   PRODUCT_TYPE[1].Motion.Ring_Turntable_Axis_2.Position[8].Pos := 318501;
   PRODUCT_TYPE[1].Motion.Ring_Turntable_Axis_2.Position[8].Vel := 10000;
   PRODUCT_TYPE[2].Motion.Ring_Turntable_Axis_2.Position[8].Pos := 318501;
   PRODUCT_TYPE[2].Motion.Ring_Turntable_Axis_2.Position[8].Vel := 10000;
   PRODUCT_TYPE[3].Motion.Ring_Turntable_Axis_2.Position[8].Pos := 318501;
   PRODUCT_TYPE[3].Motion.Ring_Turntable_Axis_2.Position[8].Vel := 10000;
   PRODUCT_TYPE[4].Motion.Ring_Turntable_Axis_2.Position[8].Pos := 318501;
   PRODUCT_TYPE[4].Motion.Ring_Turntable_Axis_2.Position[8].Vel := 10000;
   PRODUCT_TYPE[5].Motion.Ring_Turntable_Axis_2.Position[8].Pos := 318501;
   PRODUCT_TYPE[5].Motion.Ring_Turntable_Axis_2.Position[8].Vel := 10000;
   PRODUCT_TYPE[6].Motion.Ring_Turntable_Axis_2.Position[8].Pos := 318501;
   PRODUCT_TYPE[6].Motion.Ring_Turntable_Axis_2.Position[8].Vel := 10000;
   PRODUCT_TYPE[7].Motion.Ring_Turntable_Axis_2.Position[8].Pos := 318501;
   PRODUCT_TYPE[7].Motion.Ring_Turntable_Axis_2.Position[8].Vel := 10000;
   PRODUCT_TYPE[8].Motion.Ring_Turntable_Axis_2.Position[8].Pos := 318501;
   PRODUCT_TYPE[8].Motion.Ring_Turntable_Axis_2.Position[8].Vel := 10000;
   PRODUCT_TYPE[9].Motion.Ring_Turntable_Axis_2.Position[8].Pos := 318501;
   PRODUCT_TYPE[9].Motion.Ring_Turntable_Axis_2.Position[8].Vel := 10000;
   PRODUCT_TYPE[10].Motion.Ring_Turntable_Axis_2.Position[8].Pos := 318501;
   PRODUCT_TYPE[10].Motion.Ring_Turntable_Axis_2.Position[8].Vel := 10000;
   PRODUCT_TYPE[1].Motion.Ring_Turntable_Axis_2.Position[9].Pos := 0;
   PRODUCT_TYPE[1].Motion.Ring_Turntable_Axis_2.Position[9].Vel := 0;
   PRODUCT_TYPE[2].Motion.Ring_Turntable_Axis_2.Position[9].Pos := 0;
   PRODUCT_TYPE[2].Motion.Ring_Turntable_Axis_2.Position[9].Vel := 0;
   PRODUCT_TYPE[3].Motion.Ring_Turntable_Axis_2.Position[9].Pos := 0;
   PRODUCT_TYPE[3].Motion.Ring_Turntable_Axis_2.Position[9].Vel := 0;
   PRODUCT_TYPE[4].Motion.Ring_Turntable_Axis_2.Position[9].Pos := 0;
   PRODUCT_TYPE[4].Motion.Ring_Turntable_Axis_2.Position[9].Vel := 0;
   PRODUCT_TYPE[5].Motion.Ring_Turntable_Axis_2.Position[9].Pos := 0;
   PRODUCT_TYPE[5].Motion.Ring_Turntable_Axis_2.Position[9].Vel := 0;
   PRODUCT_TYPE[6].Motion.Ring_Turntable_Axis_2.Position[9].Pos := 0;
   PRODUCT_TYPE[6].Motion.Ring_Turntable_Axis_2.Position[9].Vel := 0;
   PRODUCT_TYPE[7].Motion.Ring_Turntable_Axis_2.Position[9].Pos := 0;
   PRODUCT_TYPE[7].Motion.Ring_Turntable_Axis_2.Position[9].Vel := 0;
   PRODUCT_TYPE[8].Motion.Ring_Turntable_Axis_2.Position[9].Pos := 0;
   PRODUCT_TYPE[8].Motion.Ring_Turntable_Axis_2.Position[9].Vel := 0;
   PRODUCT_TYPE[9].Motion.Ring_Turntable_Axis_2.Position[9].Pos := 0;
   PRODUCT_TYPE[9].Motion.Ring_Turntable_Axis_2.Position[9].Vel := 0;
   PRODUCT_TYPE[10].Motion.Ring_Turntable_Axis_2.Position[9].Pos := 0;
   PRODUCT_TYPE[10].Motion.Ring_Turntable_Axis_2.Position[9].Vel := 0;
   PRODUCT_TYPE[1].Motion.Ring_Turntable_Axis_2.Position[10].Pos := 0;
   PRODUCT_TYPE[1].Motion.Ring_Turntable_Axis_2.Position[10].Vel := 0;
   PRODUCT_TYPE[2].Motion.Ring_Turntable_Axis_2.Position[10].Pos := 0;
   PRODUCT_TYPE[2].Motion.Ring_Turntable_Axis_2.Position[10].Vel := 0;
   PRODUCT_TYPE[3].Motion.Ring_Turntable_Axis_2.Position[10].Pos := 0;
   PRODUCT_TYPE[3].Motion.Ring_Turntable_Axis_2.Position[10].Vel := 0;
   PRODUCT_TYPE[4].Motion.Ring_Turntable_Axis_2.Position[10].Pos := 0;
   PRODUCT_TYPE[4].Motion.Ring_Turntable_Axis_2.Position[10].Vel := 0;
   PRODUCT_TYPE[5].Motion.Ring_Turntable_Axis_2.Position[10].Pos := 0;
   PRODUCT_TYPE[5].Motion.Ring_Turntable_Axis_2.Position[10].Vel := 0;
   PRODUCT_TYPE[6].Motion.Ring_Turntable_Axis_2.Position[10].Pos := 0;
   PRODUCT_TYPE[6].Motion.Ring_Turntable_Axis_2.Position[10].Vel := 0;
   PRODUCT_TYPE[7].Motion.Ring_Turntable_Axis_2.Position[10].Pos := 0;
   PRODUCT_TYPE[7].Motion.Ring_Turntable_Axis_2.Position[10].Vel := 0;
   PRODUCT_TYPE[8].Motion.Ring_Turntable_Axis_2.Position[10].Pos := 0;
   PRODUCT_TYPE[8].Motion.Ring_Turntable_Axis_2.Position[10].Vel := 0;
   PRODUCT_TYPE[9].Motion.Ring_Turntable_Axis_2.Position[10].Pos := 0;
   PRODUCT_TYPE[9].Motion.Ring_Turntable_Axis_2.Position[10].Vel := 0;
   PRODUCT_TYPE[10].Motion.Ring_Turntable_Axis_2.Position[10].Pos := 0;
   PRODUCT_TYPE[10].Motion.Ring_Turntable_Axis_2.Position[10].Vel := 0;
   PRODUCT_TYPE[1].Motion.Ring_Turntable_Axis_2.Position[11].Pos := 0;
   PRODUCT_TYPE[1].Motion.Ring_Turntable_Axis_2.Position[11].Vel := 0;
   PRODUCT_TYPE[2].Motion.Ring_Turntable_Axis_2.Position[11].Pos := 0;
   PRODUCT_TYPE[2].Motion.Ring_Turntable_Axis_2.Position[11].Vel := 0;
   PRODUCT_TYPE[3].Motion.Ring_Turntable_Axis_2.Position[11].Pos := 0;
   PRODUCT_TYPE[3].Motion.Ring_Turntable_Axis_2.Position[11].Vel := 0;
   PRODUCT_TYPE[4].Motion.Ring_Turntable_Axis_2.Position[11].Pos := 0;
   PRODUCT_TYPE[4].Motion.Ring_Turntable_Axis_2.Position[11].Vel := 0;
   PRODUCT_TYPE[5].Motion.Ring_Turntable_Axis_2.Position[11].Pos := 0;
   PRODUCT_TYPE[5].Motion.Ring_Turntable_Axis_2.Position[11].Vel := 0;
   PRODUCT_TYPE[6].Motion.Ring_Turntable_Axis_2.Position[11].Pos := 0;
   PRODUCT_TYPE[6].Motion.Ring_Turntable_Axis_2.Position[11].Vel := 0;
   PRODUCT_TYPE[7].Motion.Ring_Turntable_Axis_2.Position[11].Pos := 0;
   PRODUCT_TYPE[7].Motion.Ring_Turntable_Axis_2.Position[11].Vel := 0;
   PRODUCT_TYPE[8].Motion.Ring_Turntable_Axis_2.Position[11].Pos := 0;
   PRODUCT_TYPE[8].Motion.Ring_Turntable_Axis_2.Position[11].Vel := 0;
   PRODUCT_TYPE[9].Motion.Ring_Turntable_Axis_2.Position[11].Pos := 0;
   PRODUCT_TYPE[9].Motion.Ring_Turntable_Axis_2.Position[11].Vel := 0;
   PRODUCT_TYPE[10].Motion.Ring_Turntable_Axis_2.Position[11].Pos := 0;
   PRODUCT_TYPE[10].Motion.Ring_Turntable_Axis_2.Position[11].Vel := 0;
   PRODUCT_TYPE[1].Motion.Ring_Turntable_Axis_2.Position[12].Pos := 0;
   PRODUCT_TYPE[1].Motion.Ring_Turntable_Axis_2.Position[12].Vel := 0;
   PRODUCT_TYPE[2].Motion.Ring_Turntable_Axis_2.Position[12].Pos := 0;
   PRODUCT_TYPE[2].Motion.Ring_Turntable_Axis_2.Position[12].Vel := 0;
   PRODUCT_TYPE[3].Motion.Ring_Turntable_Axis_2.Position[12].Pos := 0;
   PRODUCT_TYPE[3].Motion.Ring_Turntable_Axis_2.Position[12].Vel := 0;
   PRODUCT_TYPE[4].Motion.Ring_Turntable_Axis_2.Position[12].Pos := 0;
   PRODUCT_TYPE[4].Motion.Ring_Turntable_Axis_2.Position[12].Vel := 0;
   PRODUCT_TYPE[5].Motion.Ring_Turntable_Axis_2.Position[12].Pos := 0;
   PRODUCT_TYPE[5].Motion.Ring_Turntable_Axis_2.Position[12].Vel := 0;
   PRODUCT_TYPE[6].Motion.Ring_Turntable_Axis_2.Position[12].Pos := 0;
   PRODUCT_TYPE[6].Motion.Ring_Turntable_Axis_2.Position[12].Vel := 0;
   PRODUCT_TYPE[7].Motion.Ring_Turntable_Axis_2.Position[12].Pos := 0;
   PRODUCT_TYPE[7].Motion.Ring_Turntable_Axis_2.Position[12].Vel := 0;
   PRODUCT_TYPE[8].Motion.Ring_Turntable_Axis_2.Position[12].Pos := 0;
   PRODUCT_TYPE[8].Motion.Ring_Turntable_Axis_2.Position[12].Vel := 0;
   PRODUCT_TYPE[9].Motion.Ring_Turntable_Axis_2.Position[12].Pos := 0;
   PRODUCT_TYPE[9].Motion.Ring_Turntable_Axis_2.Position[12].Vel := 0;
   PRODUCT_TYPE[10].Motion.Ring_Turntable_Axis_2.Position[12].Pos := 0;
   PRODUCT_TYPE[10].Motion.Ring_Turntable_Axis_2.Position[12].Vel := 0;
   PRODUCT_TYPE[1].Motion.Ring_Turntable_Axis_2.Position[13].Pos := 0;
   PRODUCT_TYPE[1].Motion.Ring_Turntable_Axis_2.Position[13].Vel := 0;
   PRODUCT_TYPE[2].Motion.Ring_Turntable_Axis_2.Position[13].Pos := 0;
   PRODUCT_TYPE[2].Motion.Ring_Turntable_Axis_2.Position[13].Vel := 0;
   PRODUCT_TYPE[3].Motion.Ring_Turntable_Axis_2.Position[13].Pos := 0;
   PRODUCT_TYPE[3].Motion.Ring_Turntable_Axis_2.Position[13].Vel := 0;
   PRODUCT_TYPE[4].Motion.Ring_Turntable_Axis_2.Position[13].Pos := 0;
   PRODUCT_TYPE[4].Motion.Ring_Turntable_Axis_2.Position[13].Vel := 0;
   PRODUCT_TYPE[5].Motion.Ring_Turntable_Axis_2.Position[13].Pos := 0;
   PRODUCT_TYPE[5].Motion.Ring_Turntable_Axis_2.Position[13].Vel := 0;
   PRODUCT_TYPE[6].Motion.Ring_Turntable_Axis_2.Position[13].Pos := 0;
   PRODUCT_TYPE[6].Motion.Ring_Turntable_Axis_2.Position[13].Vel := 0;
   PRODUCT_TYPE[7].Motion.Ring_Turntable_Axis_2.Position[13].Pos := 0;
   PRODUCT_TYPE[7].Motion.Ring_Turntable_Axis_2.Position[13].Vel := 0;
   PRODUCT_TYPE[8].Motion.Ring_Turntable_Axis_2.Position[13].Pos := 0;
   PRODUCT_TYPE[8].Motion.Ring_Turntable_Axis_2.Position[13].Vel := 0;
   PRODUCT_TYPE[9].Motion.Ring_Turntable_Axis_2.Position[13].Pos := 0;
   PRODUCT_TYPE[9].Motion.Ring_Turntable_Axis_2.Position[13].Vel := 0;
   PRODUCT_TYPE[10].Motion.Ring_Turntable_Axis_2.Position[13].Pos := 0;
   PRODUCT_TYPE[10].Motion.Ring_Turntable_Axis_2.Position[13].Vel := 0;
   PRODUCT_TYPE[1].Motion.Ring_Turntable_Axis_2.Position[14].Pos := 0;
   PRODUCT_TYPE[1].Motion.Ring_Turntable_Axis_2.Position[14].Vel := 0;
   PRODUCT_TYPE[2].Motion.Ring_Turntable_Axis_2.Position[14].Pos := 0;
   PRODUCT_TYPE[2].Motion.Ring_Turntable_Axis_2.Position[14].Vel := 0;
   PRODUCT_TYPE[3].Motion.Ring_Turntable_Axis_2.Position[14].Pos := 0;
   PRODUCT_TYPE[3].Motion.Ring_Turntable_Axis_2.Position[14].Vel := 0;
   PRODUCT_TYPE[4].Motion.Ring_Turntable_Axis_2.Position[14].Pos := 0;
   PRODUCT_TYPE[4].Motion.Ring_Turntable_Axis_2.Position[14].Vel := 0;
   PRODUCT_TYPE[5].Motion.Ring_Turntable_Axis_2.Position[14].Pos := 0;
   PRODUCT_TYPE[5].Motion.Ring_Turntable_Axis_2.Position[14].Vel := 0;
   PRODUCT_TYPE[6].Motion.Ring_Turntable_Axis_2.Position[14].Pos := 0;
   PRODUCT_TYPE[6].Motion.Ring_Turntable_Axis_2.Position[14].Vel := 0;
   PRODUCT_TYPE[7].Motion.Ring_Turntable_Axis_2.Position[14].Pos := 0;
   PRODUCT_TYPE[7].Motion.Ring_Turntable_Axis_2.Position[14].Vel := 0;
   PRODUCT_TYPE[8].Motion.Ring_Turntable_Axis_2.Position[14].Pos := 0;
   PRODUCT_TYPE[8].Motion.Ring_Turntable_Axis_2.Position[14].Vel := 0;
   PRODUCT_TYPE[9].Motion.Ring_Turntable_Axis_2.Position[14].Pos := 0;
   PRODUCT_TYPE[9].Motion.Ring_Turntable_Axis_2.Position[14].Vel := 0;
   PRODUCT_TYPE[10].Motion.Ring_Turntable_Axis_2.Position[14].Pos := 0;
   PRODUCT_TYPE[10].Motion.Ring_Turntable_Axis_2.Position[14].Vel := 0;
   PRODUCT_TYPE[1].Motion.Ring_Turntable_Axis_2.Position[15].Pos := 0;
   PRODUCT_TYPE[1].Motion.Ring_Turntable_Axis_2.Position[15].Vel := 0;
   PRODUCT_TYPE[2].Motion.Ring_Turntable_Axis_2.Position[15].Pos := 0;
   PRODUCT_TYPE[2].Motion.Ring_Turntable_Axis_2.Position[15].Vel := 0;
   PRODUCT_TYPE[3].Motion.Ring_Turntable_Axis_2.Position[15].Pos := 0;
   PRODUCT_TYPE[3].Motion.Ring_Turntable_Axis_2.Position[15].Vel := 0;
   PRODUCT_TYPE[4].Motion.Ring_Turntable_Axis_2.Position[15].Pos := 0;
   PRODUCT_TYPE[4].Motion.Ring_Turntable_Axis_2.Position[15].Vel := 0;
   PRODUCT_TYPE[5].Motion.Ring_Turntable_Axis_2.Position[15].Pos := 0;
   PRODUCT_TYPE[5].Motion.Ring_Turntable_Axis_2.Position[15].Vel := 0;
   PRODUCT_TYPE[6].Motion.Ring_Turntable_Axis_2.Position[15].Pos := 0;
   PRODUCT_TYPE[6].Motion.Ring_Turntable_Axis_2.Position[15].Vel := 0;
   PRODUCT_TYPE[7].Motion.Ring_Turntable_Axis_2.Position[15].Pos := 0;
   PRODUCT_TYPE[7].Motion.Ring_Turntable_Axis_2.Position[15].Vel := 0;
   PRODUCT_TYPE[8].Motion.Ring_Turntable_Axis_2.Position[15].Pos := 0;
   PRODUCT_TYPE[8].Motion.Ring_Turntable_Axis_2.Position[15].Vel := 0;
   PRODUCT_TYPE[9].Motion.Ring_Turntable_Axis_2.Position[15].Pos := 0;
   PRODUCT_TYPE[9].Motion.Ring_Turntable_Axis_2.Position[15].Vel := 0;
   PRODUCT_TYPE[10].Motion.Ring_Turntable_Axis_2.Position[15].Pos := 0;
   PRODUCT_TYPE[10].Motion.Ring_Turntable_Axis_2.Position[15].Vel := 0;
   PRODUCT_TYPE[1].Motion.Ring_Turntable_Axis_2.Position[16].Pos := 0;
   PRODUCT_TYPE[1].Motion.Ring_Turntable_Axis_2.Position[16].Vel := 0;
   PRODUCT_TYPE[2].Motion.Ring_Turntable_Axis_2.Position[16].Pos := 0;
   PRODUCT_TYPE[2].Motion.Ring_Turntable_Axis_2.Position[16].Vel := 0;
   PRODUCT_TYPE[3].Motion.Ring_Turntable_Axis_2.Position[16].Pos := 0;
   PRODUCT_TYPE[3].Motion.Ring_Turntable_Axis_2.Position[16].Vel := 0;
   PRODUCT_TYPE[4].Motion.Ring_Turntable_Axis_2.Position[16].Pos := 0;
   PRODUCT_TYPE[4].Motion.Ring_Turntable_Axis_2.Position[16].Vel := 0;
   PRODUCT_TYPE[5].Motion.Ring_Turntable_Axis_2.Position[16].Pos := 0;
   PRODUCT_TYPE[5].Motion.Ring_Turntable_Axis_2.Position[16].Vel := 0;
   PRODUCT_TYPE[6].Motion.Ring_Turntable_Axis_2.Position[16].Pos := 0;
   PRODUCT_TYPE[6].Motion.Ring_Turntable_Axis_2.Position[16].Vel := 0;
   PRODUCT_TYPE[7].Motion.Ring_Turntable_Axis_2.Position[16].Pos := 0;
   PRODUCT_TYPE[7].Motion.Ring_Turntable_Axis_2.Position[16].Vel := 0;
   PRODUCT_TYPE[8].Motion.Ring_Turntable_Axis_2.Position[16].Pos := 0;
   PRODUCT_TYPE[8].Motion.Ring_Turntable_Axis_2.Position[16].Vel := 0;
   PRODUCT_TYPE[9].Motion.Ring_Turntable_Axis_2.Position[16].Pos := 0;
   PRODUCT_TYPE[9].Motion.Ring_Turntable_Axis_2.Position[16].Vel := 0;
   PRODUCT_TYPE[10].Motion.Ring_Turntable_Axis_2.Position[16].Pos := 0;
   PRODUCT_TYPE[10].Motion.Ring_Turntable_Axis_2.Position[16].Vel := 0;
   PRODUCT_TYPE[1].Motion.Ring_Turntable_Axis_2.Position[17].Pos := 0;
   PRODUCT_TYPE[1].Motion.Ring_Turntable_Axis_2.Position[17].Vel := 0;
   PRODUCT_TYPE[2].Motion.Ring_Turntable_Axis_2.Position[17].Pos := 0;
   PRODUCT_TYPE[2].Motion.Ring_Turntable_Axis_2.Position[17].Vel := 0;
   PRODUCT_TYPE[3].Motion.Ring_Turntable_Axis_2.Position[17].Pos := 0;
   PRODUCT_TYPE[3].Motion.Ring_Turntable_Axis_2.Position[17].Vel := 0;
   PRODUCT_TYPE[4].Motion.Ring_Turntable_Axis_2.Position[17].Pos := 0;
   PRODUCT_TYPE[4].Motion.Ring_Turntable_Axis_2.Position[17].Vel := 0;
   PRODUCT_TYPE[5].Motion.Ring_Turntable_Axis_2.Position[17].Pos := 0;
   PRODUCT_TYPE[5].Motion.Ring_Turntable_Axis_2.Position[17].Vel := 0;
   PRODUCT_TYPE[6].Motion.Ring_Turntable_Axis_2.Position[17].Pos := 0;
   PRODUCT_TYPE[6].Motion.Ring_Turntable_Axis_2.Position[17].Vel := 0;
   PRODUCT_TYPE[7].Motion.Ring_Turntable_Axis_2.Position[17].Pos := 0;
   PRODUCT_TYPE[7].Motion.Ring_Turntable_Axis_2.Position[17].Vel := 0;
   PRODUCT_TYPE[8].Motion.Ring_Turntable_Axis_2.Position[17].Pos := 0;
   PRODUCT_TYPE[8].Motion.Ring_Turntable_Axis_2.Position[17].Vel := 0;
   PRODUCT_TYPE[9].Motion.Ring_Turntable_Axis_2.Position[17].Pos := 0;
   PRODUCT_TYPE[9].Motion.Ring_Turntable_Axis_2.Position[17].Vel := 0;
   PRODUCT_TYPE[10].Motion.Ring_Turntable_Axis_2.Position[17].Pos := 0;
   PRODUCT_TYPE[10].Motion.Ring_Turntable_Axis_2.Position[17].Vel := 0;
   PRODUCT_TYPE[1].Motion.Ring_Turntable_Axis_2.Position[18].Pos := 0;
   PRODUCT_TYPE[1].Motion.Ring_Turntable_Axis_2.Position[18].Vel := 0;
   PRODUCT_TYPE[2].Motion.Ring_Turntable_Axis_2.Position[18].Pos := 0;
   PRODUCT_TYPE[2].Motion.Ring_Turntable_Axis_2.Position[18].Vel := 0;
   PRODUCT_TYPE[3].Motion.Ring_Turntable_Axis_2.Position[18].Pos := 0;
   PRODUCT_TYPE[3].Motion.Ring_Turntable_Axis_2.Position[18].Vel := 0;
   PRODUCT_TYPE[4].Motion.Ring_Turntable_Axis_2.Position[18].Pos := 0;
   PRODUCT_TYPE[4].Motion.Ring_Turntable_Axis_2.Position[18].Vel := 0;
   PRODUCT_TYPE[5].Motion.Ring_Turntable_Axis_2.Position[18].Pos := 0;
   PRODUCT_TYPE[5].Motion.Ring_Turntable_Axis_2.Position[18].Vel := 0;
   PRODUCT_TYPE[6].Motion.Ring_Turntable_Axis_2.Position[18].Pos := 0;
   PRODUCT_TYPE[6].Motion.Ring_Turntable_Axis_2.Position[18].Vel := 0;
   PRODUCT_TYPE[7].Motion.Ring_Turntable_Axis_2.Position[18].Pos := 0;
   PRODUCT_TYPE[7].Motion.Ring_Turntable_Axis_2.Position[18].Vel := 0;
   PRODUCT_TYPE[8].Motion.Ring_Turntable_Axis_2.Position[18].Pos := 0;
   PRODUCT_TYPE[8].Motion.Ring_Turntable_Axis_2.Position[18].Vel := 0;
   PRODUCT_TYPE[9].Motion.Ring_Turntable_Axis_2.Position[18].Pos := 0;
   PRODUCT_TYPE[9].Motion.Ring_Turntable_Axis_2.Position[18].Vel := 0;
   PRODUCT_TYPE[10].Motion.Ring_Turntable_Axis_2.Position[18].Pos := 0;
   PRODUCT_TYPE[10].Motion.Ring_Turntable_Axis_2.Position[18].Vel := 0;
   PRODUCT_TYPE[1].Motion.Ring_Turntable_Axis_2.Position[19].Pos := 0;
   PRODUCT_TYPE[1].Motion.Ring_Turntable_Axis_2.Position[19].Vel := 0;
   PRODUCT_TYPE[2].Motion.Ring_Turntable_Axis_2.Position[19].Pos := 0;
   PRODUCT_TYPE[2].Motion.Ring_Turntable_Axis_2.Position[19].Vel := 0;
   PRODUCT_TYPE[3].Motion.Ring_Turntable_Axis_2.Position[19].Pos := 0;
   PRODUCT_TYPE[3].Motion.Ring_Turntable_Axis_2.Position[19].Vel := 0;
   PRODUCT_TYPE[4].Motion.Ring_Turntable_Axis_2.Position[19].Pos := 0;
   PRODUCT_TYPE[4].Motion.Ring_Turntable_Axis_2.Position[19].Vel := 0;
   PRODUCT_TYPE[5].Motion.Ring_Turntable_Axis_2.Position[19].Pos := 0;
   PRODUCT_TYPE[5].Motion.Ring_Turntable_Axis_2.Position[19].Vel := 0;
   PRODUCT_TYPE[6].Motion.Ring_Turntable_Axis_2.Position[19].Pos := 0;
   PRODUCT_TYPE[6].Motion.Ring_Turntable_Axis_2.Position[19].Vel := 0;
   PRODUCT_TYPE[7].Motion.Ring_Turntable_Axis_2.Position[19].Pos := 0;
   PRODUCT_TYPE[7].Motion.Ring_Turntable_Axis_2.Position[19].Vel := 0;
   PRODUCT_TYPE[8].Motion.Ring_Turntable_Axis_2.Position[19].Pos := 0;
   PRODUCT_TYPE[8].Motion.Ring_Turntable_Axis_2.Position[19].Vel := 0;
   PRODUCT_TYPE[9].Motion.Ring_Turntable_Axis_2.Position[19].Pos := 0;
   PRODUCT_TYPE[9].Motion.Ring_Turntable_Axis_2.Position[19].Vel := 0;
   PRODUCT_TYPE[10].Motion.Ring_Turntable_Axis_2.Position[19].Pos := 0;
   PRODUCT_TYPE[10].Motion.Ring_Turntable_Axis_2.Position[19].Vel := 0;
   PRODUCT_TYPE[1].Motion.Ring_Turntable_Axis_2.Position[20].Pos := 0;
   PRODUCT_TYPE[1].Motion.Ring_Turntable_Axis_2.Position[20].Vel := 0;
   PRODUCT_TYPE[2].Motion.Ring_Turntable_Axis_2.Position[20].Pos := 0;
   PRODUCT_TYPE[2].Motion.Ring_Turntable_Axis_2.Position[20].Vel := 0;
   PRODUCT_TYPE[3].Motion.Ring_Turntable_Axis_2.Position[20].Pos := 0;
   PRODUCT_TYPE[3].Motion.Ring_Turntable_Axis_2.Position[20].Vel := 0;
   PRODUCT_TYPE[4].Motion.Ring_Turntable_Axis_2.Position[20].Pos := 0;
   PRODUCT_TYPE[4].Motion.Ring_Turntable_Axis_2.Position[20].Vel := 0;
   PRODUCT_TYPE[5].Motion.Ring_Turntable_Axis_2.Position[20].Pos := 0;
   PRODUCT_TYPE[5].Motion.Ring_Turntable_Axis_2.Position[20].Vel := 0;
   PRODUCT_TYPE[6].Motion.Ring_Turntable_Axis_2.Position[20].Pos := 0;
   PRODUCT_TYPE[6].Motion.Ring_Turntable_Axis_2.Position[20].Vel := 0;
   PRODUCT_TYPE[7].Motion.Ring_Turntable_Axis_2.Position[20].Pos := 0;
   PRODUCT_TYPE[7].Motion.Ring_Turntable_Axis_2.Position[20].Vel := 0;
   PRODUCT_TYPE[8].Motion.Ring_Turntable_Axis_2.Position[20].Pos := 0;
   PRODUCT_TYPE[8].Motion.Ring_Turntable_Axis_2.Position[20].Vel := 0;
   PRODUCT_TYPE[9].Motion.Ring_Turntable_Axis_2.Position[20].Pos := 0;
   PRODUCT_TYPE[9].Motion.Ring_Turntable_Axis_2.Position[20].Vel := 0;
   PRODUCT_TYPE[10].Motion.Ring_Turntable_Axis_2.Position[20].Pos := 0;
   PRODUCT_TYPE[10].Motion.Ring_Turntable_Axis_2.Position[20].Vel := 0;
   // === Motion positions (generated from XML) END ===
END_DATA_BLOCK

